// TwinCAT 3 PLC project ProcessControl
// Title: ZigaLibs.ProcessControl
// Company: Ziga Javornik
// Author: Ziga Javornik
// ProjectVersion: 0.0.2.3
// Description: A library containing objects for process control.
// ProgramVersion: 3.1.4026.26
// libraries:
//   Tc2_Standard, * (Beckhoff Automation GmbH)
//   Tc2_System, * (Beckhoff Automation GmbH)
//   Tc2_Utilities, * (Beckhoff Automation GmbH)
//   Tc3_Module, * (Beckhoff Automation GmbH)
//   TcUnit, * (www.tcunit.org)
//   ZigaLibs.Core, * (Ziga Javornik)
// project tree:
//   SOURCE/PID/DUTs/ E_BasicPidErrorId.TcDUT, E_ControllerMode.TcDUT, ST_PID_Parameters.TcDUT, T_ControllerValue.TcDUT, T_Second.TcDUT
//   SOURCE/PID/POUs/ FB_BasicPid.TcPOU
//   SOURCE/Value deviation/ E_ValueDeviationStatus.TcDUT, FB_ValueDeviation.TcPOU, I_ValueDeviation.TcIO, I_ValueDeviationLimited.TcIO, ST_Value.TcDUT
//   / TestsTask.TcTTO
//   TESTS/ PRG_TESTS.TcPOU
//   TESTS/Test suites/ FB_BasicPid_Tests.TcPOU, FB_ValueDeviation_Tests.TcPOU
// (motion and I/O tree: see PLC project logging)
// real-time tasks:
//   TASK TestsTask: cycle T#10ms, priority 20, ADS port 350
//   TASK PlcTask: cycle T#10ms, priority 21, ADS port 351

CONFIGURATION ProcessControl
    RESOURCE PLC ON TwinCAT3
        TASK TestsTask(INTERVAL := T#10ms, PRIORITY := 20);
        PROGRAM PRG_TESTS WITH TestsTask : PRG_TESTS;
    END_RESOURCE
END_CONFIGURATION

// ---- SOURCE/PID/DUTs/E_BasicPidErrorId.TcDUT
{attribute 'qualified_only'}
{attribute 'strict'}
TYPE E_BasicPidErrorId :
(
	NO_ERROR := 0,
	INVALID_PARAMETERS := 1,
	INVALID_CYCLE_TIME := 2,
	UNKNOWN_ERROR
)UINT;
END_TYPE

// ---- SOURCE/PID/DUTs/E_ControllerMode.TcDUT
{attribute 'qualified_only'}
{attribute 'strict'}
TYPE E_ControllerMode :
(
	MANUAL,
	ACTIVE
);
END_TYPE

// ---- SOURCE/PID/DUTs/ST_PID_Parameters.TcDUT
TYPE ST_PID_Parameters :
STRUCT
	Kp						: LREAL;	// Kp - Gain
	Tn						: T_Second;	// Tn - Integral gain (s)
	Tv						: T_Second;	// Tv - Derivative gain (s)
	Td						: T_Second;	// Td - Derivative damping time (s)
	CycleTime				: T_Second;	// Controller cycle time (s)
	ControllerLowerLimit	: LREAL;	// Defines the lower value of the output scaling
	ControllerUpperLimit	: LREAL;	// Defines the upper value of the output scaling
	MaxOutput				: LREAL := 100;	// Maximum output value to the controller
	(* 0-100%, when switching from manual to automatic mode controller output will only be passed 
	once it is in range of the manual setpoint. Range is defined by this parameter. 
	Setting this parameter to 0 will ommit the check and instantly activate controller (control value will most likely drop to 0!)*)
	ManualSwitchInRange	: LREAL; 
END_STRUCT
END_TYPE

// ---- SOURCE/PID/DUTs/T_ControllerValue.TcDUT
TYPE T_ControllerValue : LREAL; END_TYPE

// ---- SOURCE/PID/DUTs/T_Second.TcDUT
TYPE T_Second : LREAL; END_TYPE

// ---- SOURCE/Value deviation/E_ValueDeviationStatus.TcDUT
TYPE E_ValueDeviationStatus :
(
	OK,
	NOK
);
END_TYPE

// ---- SOURCE/Value deviation/ST_Value.TcDUT
TYPE ST_Value :
STRUCT
	Setpoint	: T_ControllerValue;
	Actual		: T_ControllerValue;
END_STRUCT
END_TYPE

// ---- SOURCE/Value deviation/I_ValueDeviation.TcIO
INTERFACE I_ValueDeviation

{attribute 'monitoring':='call'}
// Gets or sets the activation delay, before the deviation error is activated
PROPERTY ActivationDelay : TIME
GET
END_GET
SET
END_SET
END_PROPERTY

{attribute 'monitoring':='call'}
PROPERTY Enable : BOOL
GET
END_GET
SET
END_SET
END_PROPERTY

{attribute 'monitoring':='call'}
PROPERTY MaxDeviation : T_ControllerValue
GET
END_GET
SET
END_SET
END_PROPERTY

{attribute 'monitoring':='call'}
PROPERTY Status : E_ValueDeviationStatus
GET
END_GET
END_PROPERTY

{attribute 'monitoring':='call'}
PROPERTY Value : REFERENCE TO ST_Value
GET
END_GET
END_PROPERTY

END_INTERFACE

// ---- SOURCE/Value deviation/I_ValueDeviationLimited.TcIO
INTERFACE I_ValueDeviationLimited

{attribute 'monitoring':='call'}
// Gets or sets the activation delay, before the deviation error is activated
PROPERTY ActivationDelay : TIME
GET
END_GET
SET
END_SET
END_PROPERTY

{attribute 'monitoring':='call'}
PROPERTY Enable : BOOL
GET
END_GET
SET
END_SET
END_PROPERTY

{attribute 'monitoring':='call'}
PROPERTY MaxDeviation : T_ControllerValue
GET
END_GET
SET
END_SET
END_PROPERTY

{attribute 'monitoring':='call'}
PROPERTY Status : E_ValueDeviationStatus
GET
END_GET
END_PROPERTY

END_INTERFACE

// ---- TESTS/PRG_TESTS.TcPOU
PROGRAM INTERNAL PRG_TESTS

(* Instantiate test suites here. Naming convention for tests should be a suffix with _Tests.
Good practice for creating test methods is to end them with _test as well. *)
VAR
	ValueDeviationTests			: FB_ValueDeviation_Tests;
	BasicPidTests				: FB_BasicPid_Tests;
END_VAR

// Run tests in paralel
//TcUnit.RUN();

// Run tests in sequence, one after the other. Uncomment if required.
 TcUnit.RUN_IN_SEQUENCE();

END_PROGRAM

// ---- TESTS/Test suites/FB_ValueDeviation_Tests.TcPOU
FUNCTION_BLOCK INTERNAL FB_ValueDeviation_Tests EXTENDS FB_TestSuite
VAR_INPUT
END_VAR
VAR_OUTPUT
END_VAR
VAR
	_valueDeviation	: FB_ValueDeviation;
END_VAR

Test01_WhenDisabledStatusIsOk();
Test02_EnableWithNoDelay_ExpecteInstantError();
Test03_EnableWithDelay_ExpectErrorAfterDelayElapsed();
Test04_NoDelay_ChangeMaxDeviation_ExpectStatusAccordingToMaxValue();
Test05_StatusNOK_DisableAndExpectStatusOK();
Test06_NegativeMaxValue_ExpectTheDeviationAsAbsoluteValue();
Test07_NegativeValue();

METHOD PRIVATE Test01_WhenDisabledStatusIsOk
VAR_INPUT
END_VAR
TcUnit.TEST('Test01_WhenDisabledStatusIsOk');

_valueDeviation.Enable := FALSE;
_valueDeviation.MaxDeviation := 0;
_valueDeviation.Value.Setpoint := 100.0;
_valueDeviation.ActivationDelay := T#0S;
_valueDeviation();

AssertTrue(
	Condition := _valueDeviation.Status = E_ValueDeviationStatus.OK,
	Message := 'When disabled status should always be OK.');

TcUnit.TEST_FINISHED();
END_METHOD

METHOD Test02_EnableWithNoDelay_ExpecteInstantError
VAR_INPUT
END_VAR
TcUnit.TEST('Test02_EnableWithNoDelay_ExpecteInstantError');

_valueDeviation.Enable := TRUE;
_valueDeviation.MaxDeviation := 5;
_valueDeviation.ActivationDelay := T#0S;

_valueDeviation.Value.Setpoint := 10;
_valueDeviation.Value.Actual := 0;

_valueDeviation();

AssertTrue(
	Condition := _valueDeviation.Status = E_ValueDeviationStatus.NOK,
	Message := 'When enabled and no delay, status should be NOK when deviating over the threshold.');

_valueDeviation.Value.Setpoint := 10;
_valueDeviation.Value.Actual := 10;
_valueDeviation();

AssertTrue(
	Condition := _valueDeviation.Status = E_ValueDeviationStatus.OK,
	Message := 'When enabled and no delay, status should be OK when deviating under the threshold.');

TcUnit.TEST_FINISHED();
END_METHOD

METHOD Test03_EnableWithDelay_ExpectErrorAfterDelayElapsed : REFERENCE TO FB_Test
VAR_INPUT
END_VAR

VAR_INST
	TonDelayDeviation	: TON := (PT := T#1200MS);
	fbValueDeviation	: FB_ValueDeviation;
END_VAR
TcUnit.TEST('Test03_EnableWithDelay_ExpectErrorAfterDelayElapsed');

fbValueDeviation.Enable := TRUE;
fbValueDeviation.MaxDeviation := 0;
fbValueDeviation.Value.Setpoint := 100.0;
fbValueDeviation.Value.Actual := 50;
fbValueDeviation.ActivationDelay := T#1100MS;
fbValueDeviation();
TonDelayDeviation(IN := TRUE);

IF TonDelayDeviation.Q THEN
	AssertTrue(
	Condition := fbValueDeviation.Status = E_ValueDeviationStatus.NOK,
	Message := 'Deviation with delay after 1 second failed');

	TcUnit.TEST_FINISHED();
END_IF
END_METHOD

METHOD Test04_NoDelay_ChangeMaxDeviation_ExpectStatusAccordingToMaxValue
VAR_INPUT
END_VAR
TcUnit.TEST('Test04_NoDelay_ChangeMaxDeviation_ExpectStatusAccordingToMaxValue');

_valueDeviation.Enable := TRUE;
_valueDeviation.MaxDeviation := 100;
_valueDeviation.Value.Setpoint := 10;
_valueDeviation.Value.Actual := 2;
_valueDeviation.ActivationDelay := T#0S;
_valueDeviation();

AssertTrue(
	Condition := _valueDeviation.Status = E_ValueDeviationStatus.OK,
	Message := 'Changing threshold with no delay should instantly change status to OK when under max deviation.'
);

_valueDeviation.MaxDeviation := 5;
_valueDeviation();

AssertTrue(
	Condition := _valueDeviation.Status = E_ValueDeviationStatus.NOK,
	Message := 'Changing threshold with no delay should instantly change status to NOK when over max deviation.');

TcUnit.TEST_FINISHED();
END_METHOD

METHOD Test05_StatusNOK_DisableAndExpectStatusOK
VAR_INPUT
END_VAR
TcUnit.TEST('Test05_StatusNOK_DisableAndExpectStatusOK');

_valueDeviation.Enable := TRUE;
_valueDeviation.MaxDeviation := 0;
_valueDeviation.Value.Setpoint := 100.0;
_valueDeviation.Value.Actual := 500.0;
_valueDeviation.ActivationDelay := T#0S;
_valueDeviation();

AssertTrue(
	Condition := _valueDeviation.Status = E_ValueDeviationStatus.NOK,
	Message := 'Status should be NOK.'
);

_valueDeviation.Enable := FALSE;
_valueDeviation();

AssertTrue(
	Condition := _valueDeviation.Status = E_ValueDeviationStatus.OK,
	Message := 'When disabled status should always be OK.'
);

TcUnit.TEST_FINISHED();
END_METHOD

METHOD Test06_NegativeMaxValue_ExpectTheDeviationAsAbsoluteValue
VAR_INPUT
END_VAR
TcUnit.TEST('Test06_NegativeMaxValue_ExpectTheDeviationAsAbsoluteValue');

_valueDeviation.Enable := TRUE;
_valueDeviation.MaxDeviation := -10;
_valueDeviation.Value.Setpoint := 5;
_valueDeviation.Value.Actual := 8;
_valueDeviation.ActivationDelay := T#0S;
_valueDeviation();

AssertTrue(
	Condition := _valueDeviation.Status = E_ValueDeviationStatus.OK,
	Message := 'Expected status with set 5, act 8 and max deviation -10 is OK.');

_valueDeviation.MaxDeviation := -1;
_valueDeviation();

AssertTrue(
	Condition := _valueDeviation.Status = E_ValueDeviationStatus.NOK,
	Message := 'Expected status with set 5, act 8 and max deviation -1 is NOK.');


TcUnit.TEST_FINISHED();
END_METHOD

METHOD Test07_NegativeValue
VAR_INPUT
END_VAR
TcUnit.TEST('Test07_NegativeValue');

_valueDeviation.Enable := TRUE;
_valueDeviation.MaxDeviation := 10;
_valueDeviation.Value.Setpoint := -5;
_valueDeviation.Value.Actual := 0;
_valueDeviation.ActivationDelay := T#0S;
_valueDeviation();

AssertTrue(
	Condition := _valueDeviation.Status = E_ValueDeviationStatus.OK,
	Message := ' Expected status with set value -5, actual 0 and max deviation 10 is OK.');

_valueDeviation.Value.Setpoint := -15;
_valueDeviation();

AssertTrue(
	Condition := _valueDeviation.Status = E_ValueDeviationStatus.NOK,
	Message := 'Expected status with set value -15, actual 0 and max deviation 10 is NOK.');


TcUnit.TEST_FINISHED();
END_METHOD

END_FUNCTION_BLOCK

// ---- SOURCE/Value deviation/FB_ValueDeviation.TcPOU
FUNCTION_BLOCK FB_ValueDeviation IMPLEMENTS I_ValueDeviation, I_ValueDeviationLimited

VAR
	_delayDeviation		: Tc2_Standard.TON;
	_value				: ST_Value;
	_status				: E_ValueDeviationStatus;
	_maxDeviation		: T_ControllerValue;
	_enable				: BOOL;
	_activationDelay	: TIME;
END_VAR

IF _enable THEN
	_delayDeviation(
	IN := ABS(_value.Setpoint - _value.Actual) > ABS(_maxDeviation), 
	PT := _activationDelay);
ELSE
	_delayDeviation(IN := FALSE);
END_IF

IF _delayDeviation.Q THEN
	_status := E_ValueDeviationStatus.NOK;
ELSE
	_status := E_ValueDeviationStatus.OK;
END_IF

{attribute 'monitoring':='call'}
(* Gets or sets the activation delay, before the deviation error is activated*)
PROPERTY ActivationDelay : TIME
GET
ActivationDelay := _activationDelay;
END_GET
SET
_activationDelay := ActivationDelay;
END_SET
END_PROPERTY

{attribute 'monitoring':='call'}
PROPERTY Enable : BOOL
GET
Enable := _enable;
END_GET
SET
_enable := Enable;
END_SET
END_PROPERTY

{attribute 'monitoring' := 'call'}
PROPERTY MaxDeviation : T_ControllerValue
GET
MaxDeviation := _maxDeviation;
END_GET
SET
_maxDeviation := MaxDeviation;
END_SET
END_PROPERTY

{attribute 'monitoring':='call'}
PROPERTY Status : E_ValueDeviationStatus
GET
Status := _status;
END_GET
END_PROPERTY

{attribute 'monitoring':='call'}
PROPERTY Value : REFERENCE TO ST_Value
GET
Value REF= _value;
END_GET
END_PROPERTY

END_FUNCTION_BLOCK

// ---- TESTS/Test suites/FB_BasicPid_Tests.TcPOU
FUNCTION_BLOCK INTERNAL FB_BasicPid_Tests EXTENDS TcUnit.FB_TestSuite
VAR_INPUT
END_VAR
VAR_OUTPUT
END_VAR
VAR
	_pid	: FB_BasicPid;
END_VAR

_pid.Parameters.ControllerLowerLimit := 0.0;
_pid.Parameters.ControllerUpperLimit := 1000.0;
_pid.Parameters.MaxOutput := 100.0;
_pid.Parameters.CycleTime := 0.01;

Test01_ManualMode_ExpectNoPidResponse();
Test02_SwitchToActive_ExpectNoChangeUntilPidInRange();
Test03_P_Controller();
Test04_PI_Controller_ExpectIntegralAddition();

METHOD Test01_ManualMode_ExpectNoPidResponse

VAR CONSTANT
	setpointBeforeOverrange	: LREAL := 20;
	setpointAfterOverrange	: LREAL := 50;
	maxDelta				: LREAL := 0.1;
END_VAR
IF TcUnit.TEST_ORDERED('Test01_ManualMode_ExpectNoPidResponse') THEN
	_pid.Mode := E_ControllerMode.MANUAL;
	_pid.enable := TRUE;
	
	// Go under 100%, expect normal response
	_pid(manualSetpoint := setpointBeforeOverrange);
	AssertEquals_LREAL(
		Actual := _pid.output,
		Expected := setpointBeforeOverrange,
		Delta := maxDelta,
		Message := 'When in manual mode, and value is under Parameters.MaxOutput, output should be equal to manualSetpoint.');
		
	// go over 100% expected result
	_pid(manualSetpoint := _pid.Parameters.MaxOutput + 20.0);
	AssertEquals_LREAL(
		Actual := _pid.output,
		Expected := _pid.Parameters.MaxOutput,
		Delta := maxDelta,
		Message := 'When in manual mode and manualSetpoint is over the Parameters.MaxOutput parameter value, the output should be limited at Parameters.MaxOutput.');

	// Go under 100%, expect normal response
	_pid(manualSetpoint := setpointAfterOverrange);
	AssertEquals_LREAL(
		Actual := _pid.output,
		Expected := setpointAfterOverrange,
		Delta := maxDelta,
		Message := 'When in manual mode, and value is under Parameters.MaxOutput, output should be equal to manualSetpoint.');
	
	TcUnit.TEST_FINISHED();
END_IF
END_METHOD

METHOD Test02_SwitchToActive_ExpectNoChangeUntilPidInRange
VAR_INST
	iter			: UINT;
	inRangeCycles	: INT;
	valueReached	: BOOL;
END_VAR
VAR
	currentControllerOutput	: LREAL;
END_VAR
IF TcUnit.TEST_ORDERED('Test02_SwitchToActive_ExpectNoChangeUntilPidInRange') THEN
	_pid(manualSetpoint := 50);
	_pid.Parameters.Kp := 1;
	_pid.Parameters.ManualSwitchInRange := 3.0;
	_pid.Mode := E_ControllerMode.ACTIVE;
	_pid(setpoint := 800, feedback := 500 - MIN((iter * 30),500));
	
	currentControllerOutput := 100.0 * (_pid._basicPid.fCtrlOutput/_pid.Parameters.ControllerUpperLimit);
	IF ABS(currentControllerOutput - _pid.manualSetpoint) > _pid.Parameters.ManualSwitchInRange AND NOT valueReached THEN
		AssertEquals_LREAL(
			Actual := _pid.output,
			Expected := _pid.manualSetpoint,
			Delta := 0.01,
			Message := 'When switching to active mode, output should not change until internal PID reached the threshold!');
	ELSE
		inRangeCycles := inRangeCycles + 1;
		valueReached := TRUE;
		AssertEquals_LREAL(
			Actual := _pid.output,
			Expected := currentControllerOutput,
			Delta := 0.01,
			Message := 'After controller reached the threshold, output should ALWAYS follow the PID output value.');
			
		IF inRangeCycles >=5 THEN
			TcUnit.TEST_FINISHED();				
		END_IF
	END_IF
	iter := iter + 1;
END_IF
END_METHOD

METHOD PRIVATE Test03_P_Controller
VAR_INPUT
END_VAR

VAR_INST
	controller	: FB_BasicPid;
END_VAR

VAR
	expectedResult	: LREAL;
END_VAR
IF TcUnit.TEST_ORDERED('Test03_P_Controller') THEN
	// Gain of 1, expect difference in percentage
	controller.Parameters.Kp := 1.0;
	controller.Parameters.Td := 0.0;
	controller.Parameters.Tn := 0.0;
	controller.Parameters.Tv := 0.0;
	controller.Parameters.CycleTime := 0.01;
	controller.Parameters.ControllerLowerLimit := 0;
	controller.Parameters.ControllerUpperLimit := 1000.0;
	
	controller.Mode := E_ControllerMode.ACTIVE;
	controller(
		enable := TRUE,
		setpoint := 200,
		feedback := 100);
		
	expectedResult := controller.Parameters.MaxOutput * controller.Parameters.Kp * ((controller.setpoint - controller.feedback) / controller.Parameters.ControllerUpperLimit);
	AssertEquals_LREAL(
		Actual := controller.output,
		Expected := expectedResult,
		Delta := 0.1,
		Message := 'P controller output should be equal to Kp * (setpoint - actual) and scaled to limits.');
		
	// Gain of 2 - expect double result
	controller.Parameters.Kp := 2.0;
	controller.Parameters.Td := 0.0;
	controller.Parameters.Tn := 0.0;
	controller.Parameters.Tv := 0.0;
	controller.Parameters.ControllerLowerLimit := 0;
	controller.Parameters.ControllerUpperLimit := 1000.0;
	
	controller.Mode := E_ControllerMode.ACTIVE;
	controller(
		enable := TRUE,
		setpoint := 200,
		feedback := 100);
		
	expectedResult := controller.Parameters.MaxOutput * controller.Parameters.Kp * ((controller.setpoint - controller.feedback) / controller.Parameters.ControllerUpperLimit);
	AssertEquals_LREAL(
		Actual := controller.output,
		Expected := expectedResult,
		Delta := 0.1,
		Message := 'P controller output should be equal to Kp * (setpoint - actual) and scaled to limits.');
		
	TcUnit.TEST_FINISHED();
END_IF
END_METHOD

METHOD PRIVATE Test04_PI_Controller_ExpectIntegralAddition
VAR_INPUT
END_VAR

VAR_INST
	controller			: FB_BasicPid;
	testTimer			: Tc2_Standard.TON := (PT := T#1S);
	errorCount			: UINT;
	iteration			: UINT := 1;
	firstCalculation	: BOOL := TRUE;
	expectedResult		: LREAL;
	part_I				: LREAL;
	testCase			: UINT;
		
END_VAR

VAR
	part_P			: LREAL;
	sb				: ZigaLibs_Core.FB_StringBuilder;
END_VAR
IF TcUnit.TEST_ORDERED('Test04_PI_Controller_ExpectIntegralAddition') THEN
	controller.Mode := E_ControllerMode.ACTIVE;
	
	CASE testCase OF
		0:
			controller.Parameters.Kp := 1.0;
			controller.Parameters.Td := 0.0;
			controller.Parameters.Tv := 0.0;
			controller.Parameters.Tn := 0.01;
			controller.Parameters.CycleTime := 0.01;
			controller.Parameters.ControllerLowerLimit := 0;
			controller.Parameters.ControllerUpperLimit := 1000.0;
			IF testTimer.Q THEN
				part_I := 0;
				firstCalculation := TRUE;
				controller(enable := FALSE);
				testCase := testCase + 1;
				RETURN;
			END_IF
		
		1:
			controller.Parameters.Kp := 2.0;
			controller.Parameters.Td := 0.0;
			controller.Parameters.Tv := 0.0;
			controller.Parameters.Tn := 0.01;
			controller.Parameters.CycleTime := 0.01;
			controller.Parameters.ControllerLowerLimit := 0;
			controller.Parameters.ControllerUpperLimit := 1000.0;
			IF testTimer.Q THEN
				part_I := 0;
				firstCalculation := TRUE;
				controller(enable := FALSE);
				testCase := testCase + 1;
				RETURN;
			END_IF
			
		2:
			controller.Parameters.Kp := 1.0;
			controller.Parameters.Td := 0.0;
			controller.Parameters.Tv := 0.0;
			controller.Parameters.Tn := 0.1;
			controller.Parameters.CycleTime := 0.01;
			controller.Parameters.ControllerLowerLimit := 0;
			controller.Parameters.ControllerUpperLimit := 1000.0;
			IF testTimer.Q THEN
				part_I := 0;
				firstCalculation := TRUE;
				controller(enable := FALSE);
				testCase := testCase + 1;
				RETURN;
			END_IF
			
		3:			
			controller.Parameters.Kp := 2.0;
			controller.Parameters.Td := 0.0;
			controller.Parameters.Tv := 0.0;
			controller.Parameters.Tn := 0.1;
			controller.Parameters.CycleTime := 0.01;
			controller.Parameters.ControllerLowerLimit := 0;
			controller.Parameters.ControllerUpperLimit := 1000.0;
			IF testTimer.Q THEN
				TcUnit.TEST_FINISHED();
			END_IF
	END_CASE
	
	testTimer(IN := NOT testTimer.Q);
	
	controller(
		enable := TRUE,
		setpoint := 300,
		feedback := 100);

	part_P := (controller.setpoint - controller.feedback)/controller.Parameters.ControllerUpperLimit;
	part_I := part_I +  ((1/controller.Parameters.Tn) * (controller.setpoint - controller.feedback) / (controller.Parameters.ControllerUpperLimit * 100.0));
	
	IF firstCalculation THEN
		part_I := part_I / 2; 
	END_IF
	
	expectedResult := MIN(
		controller.Parameters.MaxOutput,
		controller.Parameters.MaxOutput * controller.Parameters.Kp * (part_P + part_I));
	
	IF expectedResult <> controller.output THEN
		errorCount := errorCount + 1;
	END_IF

	AssertEquals_LREAL(
		Actual := controller.output,
		Expected := expectedResult,
		Delta := 0.1,
		Message := sb.AddString('P controller output should be equal to Kp * (setpoint - actual) and scaled to limits. Count: ')
					.AddAny(errorCount)
					.AddString('Parameteres: ')
					.AddString('[Kp=').AddAny(controller.Parameters.Kp)
					.AddString('][Tn=').AddAny(controller.Parameters.Tn).AddString('s]')
					.Create());
		
	firstCalculation := FALSE;
	iteration := iteration + 1;
END_IF
END_METHOD

END_FUNCTION_BLOCK

// ---- SOURCE/PID/POUs/FB_BasicPid.TcPOU
// A discretized PID element. Transfer function:
// G(s) = Kp*(1+ (1/(Tn)) + (Tv/(1+Td)) )
FUNCTION_BLOCK FB_BasicPid EXTENDS ZigaLibs_Core.FB_HasTaskInfo
VAR_INPUT
	enable			: BOOL;		// Enables PID
	setpoint		: LREAL;	// Setpoint for PID controller when in ACTIVE moed
	manualSetpoint	: LREAL;	// Setpoint passed to output when MANUAL mode is active
	feedback		: LREAL;	// Feedback value for PID
	reset			: BOOL;		// Resets the controller
END_VAR
VAR_OUTPUT
	output	: LREAL;	// Output for the control variable, spanning from 0-100 (%) betwee Parameters.Minimum
	error	: BOOL;		// TRUE if error (incorrect parameters)
	errorId	: E_BasicPidErrorId;
END_VAR
VAR
	_parameters					: ST_PID_Parameters;
	_basicPid					: Tc2_Utilities.FB_BasicPID;
	_mode						: E_ControllerMode := E_ControllerMode.ACTIVE;
	_taskTimeAsSeconds			: LREAL;
	_modeChanged				: BOOL;
	_waitForControllerInRange	: BOOL;
	_setpointFromManualMode		: LREAL;
	_percentValueCurrent		: LREAL;
	_output						: LREAL;
END_VAR

error := FALSE;
IF THIS^.TaskInfo.CycleTime <> 0 THEN
	_taskTimeAsSeconds := 1000.0/DINT_TO_LREAL(THIS^.TaskInfo.CycleTime);	
END_IF


_basicPid.fKp := _parameters.Kp;
_basicPid.fTn := _parameters.Tn;
_basicPid.fTd := _parameters.Td;
_basicPid.fTv := _parameters.Tv;

IF _basicPid.fCtrlCycleTime = 0 OR (_parameters.CycleTime < _taskTimeAsSeconds) THEN
	IF _taskTimeAsSeconds <> 0 THEN
		// Set control time to a minimum of task cycle time
		_basicPid.fCtrlCycleTime := _taskTimeAsSeconds;
	ELSE
		// Cycle time invalid and can't be determined - exit
		errorId := E_BasicPidErrorId.INVALID_CYCLE_TIME;
		error := TRUE;
		output := 0;
		RETURN;
	END_IF
END_IF


IF NOT enable THEN
	_basicPid(
		bReset := NOT _basicPid.bReset, 
		fSetpointValue := 0, 
		fActualValue := 0);
	_output := 0;
	_waitForControllerInRange := FALSE;
ELSE
	CASE _mode OF
		E_ControllerMode.MANUAL:
			_output := MIN(_parameters.MaxOutput, MAX(0, manualSetpoint));
			_setpointFromManualMode := _output;
			_basicPid(
				bReset := NOT _basicPid.bReset, 
				fSetpointValue := 0, 
				fActualValue := 0);
		
		E_ControllerMode.ACTIVE:
			IF _modeChanged THEN
				_waitForControllerInRange := manualSetpoint <> 0;
			END_IF
			
			_basicPid(
				fActualValue := feedback,
				fSetpointValue := setpoint,
				bReset := FALSE);
				
			_percentValueCurrent := THIS^.ValueToPercentage(_basicPid.fCtrlOutput);
			
			// Wait for controller to reach the manual setpoint before activating it
			IF _waitForControllerInRange AND _parameters.ManualSwitchInRange <> 0.0 THEN
				IF (_percentValueCurrent + _parameters.ManualSwitchInRange) >= _setpointFromManualMode  THEN
					// Controller has reached the manual setpoint. Reset flag and instantly pass the value to output.
					_waitForControllerInRange := FALSE;
					_output := THIS^.ValueToPercentage(_basicPid.fCtrlOutput);
				ELSE
					// Wait for controller to reach the manual setpoint. Pass the last manual value until then.
					_output := _setpointFromManualMode;
				END_IF
			ELSE
				// Controller has reached the setpoint or the threshold is 0 - output is controlled by the PID
				_output := THIS^.ValueToPercentage(_basicPid.fCtrlOutput);
			END_IF
	END_CASE
END_IF

error := error OR _basicPid.nErrorStatus <> E_BasicPidErrorId.NO_ERROR;

CASE _basicPid.nErrorStatus OF
	0:
		errorId := E_BasicPidErrorId.NO_ERROR;
	1:
		errorId := E_BasicPidErrorId.INVALID_PARAMETERS;
	2:
		errorId := E_BasicPidErrorId.INVALID_CYCLE_TIME;
	ELSE
		errorId := E_BasicPidErrorId.UNKNOWN_ERROR;
END_CASE

output := _output;
_modeChanged := FALSE;

PROPERTY Mode : E_ControllerMode
GET
Mode := _mode;
END_GET
SET
IF _mode <> Mode THEN
	_modeChanged := TRUE;
END_IF

_mode := Mode;
END_SET
END_PROPERTY

{attribute 'monitoring' := 'variable'}
PROPERTY Parameters : REFERENCE TO ST_PID_Parameters
GET
Parameters REF= _parameters;
END_GET
SET
_parameters := Parameters;
END_SET
END_PROPERTY

// Calculates the percentage. Negative values are ommited and 0 is returned. Output is limited to _parameters.MaxOutput.
METHOD PRIVATE ValueToPercentage : LREAL
VAR_INPUT
	value	: LREAL;
END_VAR

VAR
	rangeSpan	: LREAL;
END_VAR
rangeSpan := (_parameters.ControllerUpperLimit - _parameters.ControllerLowerLimit);
IF value <= _parameters.ControllerLowerLimit OR rangeSpan <= 0THEN
	ValueToPercentage := 0.0;
	RETURN;
END_IF

ValueToPercentage := MIN((100.0 * (value / rangeSpan)), _parameters.MaxOutput);
END_METHOD

END_FUNCTION_BLOCK
